// Device/Application/POUs/FB_MasterOperatorControl
FUNCTION_BLOCK FB_MasterOperatorControl
VAR_INPUT
    xAutoModeSelected     : BOOL;
    xEmergencyStopHealthy : BOOL;
    xFactoryIORunning     : BOOL;
    xManualModeSelected   : BOOL;
    xPlantFaulted         : BOOL;
    xResetPB              : BOOL;
    xStartPB              : BOOL;
    xStopCircuitHealthy   : BOOL;
END_VAR
VAR_OUTPUT
    xAutoModeActive   : BOOL;
    xAutoRun          : BOOL;
    xEnable           : BOOL;
    xManualModeActive : BOOL;
    xResetPulse       : BOOL;
    xResetRequired    : BOOL := TRUE;
    xRunLatched       : BOOL;
    xStopPending      : BOOL;
END_VAR
VAR
    fbResetEdge    : R_TRIG;
    fbStartEdge    : R_TRIG;
    xModeValid     : BOOL;
    xSafetyHealthy : BOOL;
END_VAR

// Convert the MASTER push buttons into one-scan events.
fbResetEdge(CLK := xResetPB);
fbStartEdge(CLK := xStartPB);

// Exactly one MASTER operating mode must be selected.
xModeValid :=
    xAutoModeSelected XOR xManualModeSelected;

xAutoModeActive :=
    xAutoModeSelected
    AND NOT xManualModeSelected;

xManualModeActive :=
    xManualModeSelected
    AND NOT xAutoModeSelected;

// MASTER safety availability.
// The ordinary Stop circuit is handled separately so Auto mode
// can finish its current transaction under controlled-stop logic.
xSafetyHealthy :=
    xEmergencyStopHealthy
    AND xFactoryIORunning
    AND xModeValid;

// One-scan default.
xResetPulse := FALSE;

// Immediate safety loss cancels all MASTER authority.
IF NOT xSafetyHealthy THEN
    xResetRequired := TRUE;
    xRunLatched := FALSE;
    xStopPending := FALSE;

// Reset has priority over a latched plant fault so that the
// coordinator can actually receive the reset pulse.
ELSIF fbResetEdge.Q AND xStopCircuitHealthy THEN
    xResetPulse := TRUE;
    xResetRequired := FALSE;
    xRunLatched := FALSE;
    xStopPending := FALSE;

// A plant fault removes the run latch and requires acknowledgement.
ELSIF xPlantFaulted THEN
    xResetRequired := TRUE;
    xRunLatched := FALSE;
    xStopPending := FALSE;

// MASTER Stop requests controlled completion in Auto mode.
ELSIF NOT xStopCircuitHealthy THEN
    IF xRunLatched THEN
        xStopPending := TRUE;
    END_IF

    xRunLatched := FALSE;

// Selecting Manual removes automatic authority.
// Local unit panels will receive authority in a later step.
ELSIF xManualModeActive THEN
    IF xRunLatched THEN
        xStopPending := TRUE;
    END_IF

    xRunLatched := FALSE;

// MASTER Start is accepted only in Auto after a valid reset.
ELSIF fbStartEdge.Q
    AND xAutoModeActive
    AND NOT xResetRequired
THEN
    xRunLatched := TRUE;
    xStopPending := FALSE;
END_IF

xAutoRun :=
    xAutoModeActive
    AND xRunLatched;

// Manual mode requires a healthy MASTER Stop circuit.
// Auto mode retains enable during a controlled-stop request.
xEnable :=
    xSafetyHealthy
    AND NOT xPlantFaulted
    AND NOT xResetRequired
    AND (
        xAutoModeActive
        OR xStopCircuitHealthy
    );

END_FUNCTION_BLOCK

// Device/Application/POUs/FB_PackoutCarrierStation
FUNCTION_BLOCK FB_PackoutCarrierStation
VAR_INPUT
    tStepTimeout      : TIME := T#30S;
    xCarrierReq       : BOOL;
    xDownstreamAck    : BOOL;
    xDownstreamReady  : BOOL;
    xEnable           : BOOL;
    xLoadComplete     : BOOL;
    xPalletAtLoad     : BOOL;
    xProductLoaded    : BOOL;
    xReset            : BOOL;
	xRun 			  : BOOL;
END_VAR
VAR_OUTPUT
    eState                    : E_PackoutCarrierState :=
                                    E_PackoutCarrierState.Stopped;
    uiFaultCode               : UINT;
    xBusy                     : BOOL;
    xCarrierConveyorCmd       : BOOL;
    xCarrierEmitterCmd        : BOOL;
    xCarrierInfeedConveyorCmd : BOOL;
    xCarrierReady             : BOOL;
    xFaulted                  : BOOL;
    xLoadAccepted             : BOOL;
    xLoadedCarrierReq         : BOOL;
    xReady                    : BOOL;
END_VAR
VAR
    ePreviousState 	   : E_PackoutCarrierState :=
                         E_PackoutCarrierState.Stopped;
	fbCarrierEmitPulse : TP;
    fbStepTimeout 	   : TON;
	xCarrierEmitIssued : BOOL;
    xStateChanged  	   : BOOL;
    xTimedState    	   : BOOL;
END_VAR

// Detect state transitions.
xStateChanged := eState <> ePreviousState;

fbCarrierEmitPulse(
    IN :=
        xEnable
        AND xRun
        AND NOT xCarrierEmitIssued
        AND
        (eState = E_PackoutCarrierState.FeedingCarrier)
        AND NOT xPalletAtLoad,
    PT := T#500MS
);

// Remember that this carrier has already been emitted.
// Preserve this latch across a controlled Stop.
IF fbCarrierEmitPulse.Q THEN
    xCarrierEmitIssued := TRUE;
END_IF

// Arrival proves that another carrier may be emitted later.
IF xPalletAtLoad THEN
    xCarrierEmitIssued := FALSE;
END_IF

xTimedState :=
    (eState = E_PackoutCarrierState.FeedingCarrier)
    OR
    (eState = E_PackoutCarrierState.TransferringCarrier)
    OR
    (eState =
        E_PackoutCarrierState.WaitingForDownstreamAckClear);

fbStepTimeout(
    IN :=
        xEnable
        AND xRun
        AND xTimedState
        AND NOT xStateChanged,
    PT := tStepTimeout
);

ePreviousState := eState;

// Safe physical-output defaults.
xCarrierConveyorCmd := FALSE;
xCarrierEmitterCmd := FALSE;
xCarrierInfeedConveyorCmd := FALSE;

IF xReset THEN
    eState := E_PackoutCarrierState.Stopped;
    ePreviousState := E_PackoutCarrierState.Stopped;
    uiFaultCode := 0;

ELSIF xEnable AND xRun THEN
    CASE eState OF

        E_PackoutCarrierState.Stopped:
            uiFaultCode := 0;
            eState :=
                E_PackoutCarrierState.WaitingForCarrierRequest;


        E_PackoutCarrierState.WaitingForCarrierRequest:
            IF xPalletAtLoad THEN
                eState :=
                    E_PackoutCarrierState.HoldingCarrierAtLoad;

            ELSIF xCarrierReq THEN
                eState :=
                    E_PackoutCarrierState.FeedingCarrier;
            END_IF


        E_PackoutCarrierState.FeedingCarrier:
            xCarrierConveyorCmd := TRUE;
            xCarrierEmitterCmd := fbCarrierEmitPulse.Q;
            xCarrierInfeedConveyorCmd := TRUE;

            IF xPalletAtLoad THEN
                eState :=
                    E_PackoutCarrierState.HoldingCarrierAtLoad;

            ELSIF fbStepTimeout.Q THEN
                uiFaultCode := 601;
                eState := E_PackoutCarrierState.Faulted;
            END_IF


        E_PackoutCarrierState.HoldingCarrierAtLoad:
            IF NOT xPalletAtLoad THEN
                IF xCarrierReq THEN
                    eState :=
                        E_PackoutCarrierState.FeedingCarrier;
                ELSE
                    eState :=
                        E_PackoutCarrierState
                            .WaitingForCarrierRequest;
                END_IF

            ELSIF xLoadComplete AND xProductLoaded THEN
                eState :=
                    E_PackoutCarrierState
                        .RequestingPlantStorage;
            END_IF


        E_PackoutCarrierState.RequestingPlantStorage:
            // Do not move until the loader has cleared its
            // LoadComplete request and Plant Storage is ready.
            IF NOT xLoadComplete AND xDownstreamReady THEN
                eState :=
                    E_PackoutCarrierState.TransferringCarrier;
            END_IF


        E_PackoutCarrierState.TransferringCarrier:
            xCarrierConveyorCmd := TRUE;

            IF xDownstreamAck THEN
                eState :=
                    E_PackoutCarrierState
                        .WaitingForDownstreamAckClear;

            ELSIF fbStepTimeout.Q THEN
                uiFaultCode := 602;
                eState := E_PackoutCarrierState.Faulted;
            END_IF


        E_PackoutCarrierState.WaitingForDownstreamAckClear:
            IF NOT xDownstreamAck THEN
                eState :=
                    E_PackoutCarrierState
                        .WaitingForCarrierRequest;

            ELSIF fbStepTimeout.Q THEN
                uiFaultCode := 603;
                eState := E_PackoutCarrierState.Faulted;
            END_IF


        E_PackoutCarrierState.Faulted:
            // Physical outputs remain at their safe defaults.


    ELSE
        uiFaultCode := 698;
        eState := E_PackoutCarrierState.Faulted;

    END_CASE
END_IF

// State-derived status and nonphysical handshakes.
xBusy :=
    (eState = E_PackoutCarrierState.FeedingCarrier)
    OR
    (eState = E_PackoutCarrierState.RequestingPlantStorage)
    OR
    (eState = E_PackoutCarrierState.TransferringCarrier)
    OR
    (eState =
        E_PackoutCarrierState.WaitingForDownstreamAckClear);

xCarrierReady :=
    xPalletAtLoad
    AND
    (eState = E_PackoutCarrierState.HoldingCarrierAtLoad);

xFaulted :=
    eState = E_PackoutCarrierState.Faulted;

xLoadAccepted :=
    xLoadComplete
    AND
    (eState =
        E_PackoutCarrierState.RequestingPlantStorage);

xLoadedCarrierReq :=
    NOT xLoadComplete
    AND
    (
        (eState =
            E_PackoutCarrierState.RequestingPlantStorage)
        OR
        (eState =
            E_PackoutCarrierState.TransferringCarrier)
    );

xReady :=
    xEnable
    AND xRun
	AND
    (
        (eState =
            E_PackoutCarrierState.WaitingForCarrierRequest)
        OR
        (eState =
            E_PackoutCarrierState.HoldingCarrierAtLoad)
    );

// Faults always remove physical commands.
IF xFaulted THEN
    xCarrierConveyorCmd := FALSE;
    xCarrierEmitterCmd := FALSE;
    xCarrierInfeedConveyorCmd := FALSE;
    xCarrierReady := FALSE;
    xReady := FALSE;
END_IF

END_FUNCTION_BLOCK

// Device/Application/POUs/FB_PackoutLoader
FUNCTION_BLOCK FB_PackoutLoader
VAR_INPUT
    tStepTimeout            : TIME := T#20S;
    xCarrierReady           : BOOL;
    xEnable                 : BOOL;
    xItemDetected           : BOOL;
    xLoadAccepted           : BOOL;
    xMovingX                : BOOL;
    xMovingZ                : BOOL;
    xProductAtPick          : BOOL;
    xProductLoaded          : BOOL;
    xProductTransferPermit  : BOOL;
    xReset                  : BOOL;
	xRun                    : BOOL;
END_VAR
VAR_OUTPUT
    diProductCount          : DINT;
    eState                  : E_PackoutLoaderState :=
                                  E_PackoutLoaderState.Stopped;
    uiFaultCode             : UINT;
    xBufferConveyor1Cmd     : BOOL;
    xBufferConveyor2Cmd     : BOOL;
    xBufferConveyor3Cmd     : BOOL;
    xBusy                   : BOOL;
    xCarrierReq             : BOOL;
    xFaulted                : BOOL;
    xGrabCmd                : BOOL;
    xLoadComplete           : BOOL;
    xMoveXCmd               : BOOL;
    xMoveZCmd               : BOOL;
    xPickConveyorCmd        : BOOL;
    xProductTransferAck     : BOOL;
    xProductTransferReady   : BOOL;
    xReady                  : BOOL;
END_VAR
VAR
    ePreviousState  : E_PackoutLoaderState :=
                          E_PackoutLoaderState.Stopped;
    fbGrabSettle     : TON;
	fbHomeStable     : TON;
    fbReleaseSettle  : TON;
    fbStepTimeout    : TON;
	xProductAccepted : BOOL;
    xSawXMotion      : BOOL;
    xSawZMotion      : BOOL;
    xStateChanged    : BOOL;
    xTimedState      : BOOL;
END_VAR

// Detect state transitions.
xStateChanged := eState <> ePreviousState;

IF xStateChanged THEN
    xSawXMotion := FALSE;
    xSawZMotion := FALSE;
END_IF

IF xMovingX THEN
    xSawXMotion := TRUE;
END_IF

IF xMovingZ THEN
    xSawZMotion := TRUE;
END_IF

fbHomeStable(
    IN :=
        xEnable
        AND xRun
        AND (eState = E_PackoutLoaderState.Homing)
        AND NOT xMovingX
        AND NOT xMovingZ,
    PT := T#500MS
);

xTimedState :=
    (eState <> E_PackoutLoaderState.Stopped)
    AND (eState <> E_PackoutLoaderState.WaitingForCarrier)
    AND (eState <> E_PackoutLoaderState.WaitingForProduct)
    AND
    (eState <>
        E_PackoutLoaderState.WaitingForLoadAcceptance)
    AND (eState <> E_PackoutLoaderState.Complete)
    AND (eState <> E_PackoutLoaderState.Faulted);

fbStepTimeout(
    IN :=
        xEnable
        AND xRun
        AND xTimedState
        AND NOT xStateChanged,
    PT := tStepTimeout
);

fbGrabSettle(
    IN :=
        xEnable
        AND xRun
        AND
        (eState = E_PackoutLoaderState.GrippingProduct),
    PT := T#500MS
);

fbReleaseSettle(
    IN :=
        xEnable
        AND xRun
        AND
        (eState = E_PackoutLoaderState.ReleasingProduct),
    PT := T#500MS
);

ePreviousState := eState;

// Safe defaults.
xBufferConveyor1Cmd := FALSE;
xBufferConveyor2Cmd := FALSE;
xBufferConveyor3Cmd := FALSE;
xBusy := FALSE;
xCarrierReq := FALSE;
xGrabCmd := FALSE;
xLoadComplete := FALSE;
xMoveXCmd := FALSE;
xMoveZCmd := FALSE;
xPickConveyorCmd := FALSE;
xProductTransferAck := FALSE;
xProductTransferReady := FALSE;
xReady := FALSE;

IF xReset THEN
    diProductCount := 0;
    eState := E_PackoutLoaderState.Stopped;
    ePreviousState := E_PackoutLoaderState.Stopped;
    uiFaultCode := 0;
    xFaulted := FALSE;
    xProductAccepted := FALSE;
    xSawXMotion := FALSE;
    xSawZMotion := FALSE;

ELSIF NOT xEnable THEN
    eState := E_PackoutLoaderState.Stopped;
    ePreviousState := E_PackoutLoaderState.Stopped;
    uiFaultCode := 0;
    xFaulted := FALSE;
    xProductAccepted := FALSE;
    xSawXMotion := FALSE;
    xSawZMotion := FALSE;

ELSIF xRun THEN
    CASE eState OF

        E_PackoutLoaderState.Stopped:
            xFaulted := FALSE;
            eState := E_PackoutLoaderState.Homing;


        E_PackoutLoaderState.Homing:
            // Both monostable axes return home with commands removed.
            IF fbHomeStable.Q THEN
                eState :=
                    E_PackoutLoaderState.WaitingForCarrier;

            ELSIF fbStepTimeout.Q THEN
                uiFaultCode := 501;
                xFaulted := TRUE;
                eState := E_PackoutLoaderState.Faulted;
            END_IF


        E_PackoutLoaderState.WaitingForCarrier:
            xCarrierReq := TRUE;
            xReady := TRUE;

            IF xCarrierReady THEN
                eState :=
                    E_PackoutLoaderState.WaitingForProduct;
            END_IF


        E_PackoutLoaderState.WaitingForProduct:
            xReady := TRUE;

            IF NOT xCarrierReady THEN
                eState :=
                    E_PackoutLoaderState.WaitingForCarrier;

            ELSE
                // A product already staged at the pick sensor
                // must not withdraw the loader's readiness.
                xProductTransferReady := NOT xProductLoaded;

                IF xProductTransferPermit THEN
                    xBufferConveyor1Cmd := NOT xProductAtPick;
                    xBufferConveyor2Cmd := NOT xProductAtPick;
                    xBufferConveyor3Cmd := NOT xProductAtPick;
                    xPickConveyorCmd := NOT xProductAtPick;

                    IF xProductAtPick THEN
                        xProductAccepted := TRUE;
                        eState :=
                            E_PackoutLoaderState.MovingToProduct;
                    END_IF
                END_IF
            END_IF


        E_PackoutLoaderState.MovingToProduct:
            xBusy := TRUE;
            xMoveXCmd := TRUE;

            IF xSawXMotion AND NOT xMovingX THEN
                eState :=
                    E_PackoutLoaderState.LoweringToProduct;

            ELSIF fbStepTimeout.Q THEN
                uiFaultCode := 503;
                xFaulted := TRUE;
                eState := E_PackoutLoaderState.Faulted;
            END_IF


        E_PackoutLoaderState.LoweringToProduct:
            xBusy := TRUE;
            xMoveXCmd := TRUE;
            xMoveZCmd := TRUE;

            IF xSawZMotion AND NOT xMovingZ THEN
                eState :=
                    E_PackoutLoaderState.GrippingProduct;

            ELSIF fbStepTimeout.Q THEN
                uiFaultCode := 504;
                xFaulted := TRUE;
                eState := E_PackoutLoaderState.Faulted;
            END_IF


        E_PackoutLoaderState.GrippingProduct:
            xBusy := TRUE;
            xGrabCmd := TRUE;
            xMoveXCmd := TRUE;
            xMoveZCmd := TRUE;

            IF fbGrabSettle.Q AND xItemDetected THEN
                eState :=
                    E_PackoutLoaderState.RaisingProduct;

            ELSIF fbStepTimeout.Q THEN
                uiFaultCode := 505;
                xFaulted := TRUE;
                eState := E_PackoutLoaderState.Faulted;
            END_IF


        E_PackoutLoaderState.RaisingProduct:
            xBusy := TRUE;
            xGrabCmd := TRUE;
            xMoveXCmd := TRUE;

            IF xSawZMotion AND NOT xMovingZ THEN
                eState :=
                    E_PackoutLoaderState.MovingToCarrier;

            ELSIF fbStepTimeout.Q THEN
                uiFaultCode := 506;
                xFaulted := TRUE;
                eState := E_PackoutLoaderState.Faulted;
            END_IF


        E_PackoutLoaderState.MovingToCarrier:
            xBusy := TRUE;
            xGrabCmd := TRUE;

            // Removing the X command retracts the monostable
            // horizontal axis towards the carrier.
            IF xSawXMotion AND NOT xMovingX THEN
                eState :=
                    E_PackoutLoaderState.LoweringToCarrier;

            ELSIF fbStepTimeout.Q THEN
                uiFaultCode := 507;
                xFaulted := TRUE;
                eState := E_PackoutLoaderState.Faulted;
            END_IF


        E_PackoutLoaderState.LoweringToCarrier:
            xBusy := TRUE;
            xGrabCmd := TRUE;
            xMoveZCmd := TRUE;

            IF xSawZMotion AND NOT xMovingZ THEN
                eState :=
                    E_PackoutLoaderState.ReleasingProduct;

            ELSIF fbStepTimeout.Q THEN
                uiFaultCode := 508;
                xFaulted := TRUE;
                eState := E_PackoutLoaderState.Faulted;
            END_IF


        E_PackoutLoaderState.ReleasingProduct:
            xBusy := TRUE;
            xMoveZCmd := TRUE;

            IF fbReleaseSettle.Q AND NOT xItemDetected THEN
                eState :=
                    E_PackoutLoaderState.RaisingFromCarrier;

            ELSIF fbStepTimeout.Q THEN
                uiFaultCode := 509;
                xFaulted := TRUE;
                eState := E_PackoutLoaderState.Faulted;
            END_IF


        E_PackoutLoaderState.RaisingFromCarrier:
            xBusy := TRUE;

            IF xSawZMotion AND NOT xMovingZ THEN
                eState :=
                    E_PackoutLoaderState.ReturningHome;

            ELSIF fbStepTimeout.Q THEN
                uiFaultCode := 510;
                xFaulted := TRUE;
                eState := E_PackoutLoaderState.Faulted;
            END_IF


        E_PackoutLoaderState.ReturningHome:
            xBusy := TRUE;

            IF NOT xMovingX AND NOT xMovingZ THEN
                eState :=
                    E_PackoutLoaderState.VerifyingLoad;

            ELSIF fbStepTimeout.Q THEN
                uiFaultCode := 511;
                xFaulted := TRUE;
                eState := E_PackoutLoaderState.Faulted;
            END_IF


        E_PackoutLoaderState.VerifyingLoad:
            xBusy := TRUE;

            IF xCarrierReady AND xProductLoaded THEN
                diProductCount := diProductCount + 1;
                eState :=
                    E_PackoutLoaderState
                        .WaitingForLoadAcceptance;

            ELSIF fbStepTimeout.Q THEN
                uiFaultCode := 512;
                xFaulted := TRUE;
                eState := E_PackoutLoaderState.Faulted;
            END_IF


        E_PackoutLoaderState.WaitingForLoadAcceptance:
            xBusy := TRUE;
            xLoadComplete := TRUE;

            IF xLoadAccepted THEN
                eState := E_PackoutLoaderState.Complete;
            END_IF


        E_PackoutLoaderState.Complete:
            // Wait for the carrier station to clear acknowledgement.
            IF NOT xLoadAccepted THEN
                eState :=
                    E_PackoutLoaderState.WaitingForCarrier;
            END_IF


        E_PackoutLoaderState.Faulted:
            xFaulted := TRUE;


    ELSE
        uiFaultCode := 599;
        xFaulted := TRUE;
        eState := E_PackoutLoaderState.Faulted;

    END_CASE
END_IF

// A controlled Stop preserves the current transaction.
// The monostable axes retain the command appropriate to the
// current sequence state.
IF xEnable AND NOT xRun AND NOT xFaulted THEN
    xBusy :=
        (eState = E_PackoutLoaderState.MovingToProduct)
        OR (eState = E_PackoutLoaderState.LoweringToProduct)
        OR (eState = E_PackoutLoaderState.GrippingProduct)
        OR (eState = E_PackoutLoaderState.RaisingProduct)
        OR (eState = E_PackoutLoaderState.MovingToCarrier)
        OR (eState = E_PackoutLoaderState.LoweringToCarrier)
        OR (eState = E_PackoutLoaderState.ReleasingProduct)
        OR (eState = E_PackoutLoaderState.RaisingFromCarrier)
        OR (eState = E_PackoutLoaderState.ReturningHome)
        OR (eState = E_PackoutLoaderState.VerifyingLoad)
        OR
        (eState =
            E_PackoutLoaderState.WaitingForLoadAcceptance);

    xGrabCmd :=
        (eState = E_PackoutLoaderState.GrippingProduct)
        OR (eState = E_PackoutLoaderState.RaisingProduct)
        OR (eState = E_PackoutLoaderState.MovingToCarrier)
        OR (eState = E_PackoutLoaderState.LoweringToCarrier);

    xLoadComplete :=
        eState =
            E_PackoutLoaderState.WaitingForLoadAcceptance;

    xMoveXCmd :=
        (eState = E_PackoutLoaderState.MovingToProduct)
        OR (eState = E_PackoutLoaderState.LoweringToProduct)
        OR (eState = E_PackoutLoaderState.GrippingProduct)
        OR (eState = E_PackoutLoaderState.RaisingProduct);

    xMoveZCmd :=
        (eState = E_PackoutLoaderState.LoweringToProduct)
        OR (eState = E_PackoutLoaderState.GrippingProduct)
        OR (eState = E_PackoutLoaderState.LoweringToCarrier)
        OR (eState = E_PackoutLoaderState.ReleasingProduct);
END_IF

// Hold acknowledgement until the coordinator removes its permit.
xProductTransferAck := xProductAccepted;

IF xProductAccepted
    AND xRun
    AND NOT xProductTransferPermit
THEN
    xProductAccepted := FALSE;
    xProductTransferAck := FALSE;
END_IF

// Faults remove every command and handshake.
IF xFaulted THEN
    xBufferConveyor1Cmd := FALSE;
    xBufferConveyor2Cmd := FALSE;
    xBufferConveyor3Cmd := FALSE;
    xCarrierReq := FALSE;
    xGrabCmd := FALSE;
    xLoadComplete := FALSE;
    xMoveXCmd := FALSE;
    xMoveZCmd := FALSE;
    xPickConveyorCmd := FALSE;
    xProductAccepted := FALSE;
    xProductTransferAck := FALSE;
    xProductTransferReady := FALSE;
    xReady := FALSE;
END_IF

END_FUNCTION_BLOCK

// Device/Application/POUs/FB_PairDiverter
FUNCTION_BLOCK FB_PairDiverter
VAR_INPUT
	tLidPositionTime 		   : TIME := T#300MS;
    tStepTimeout               : TIME := T#15S;
    xAssemblyBaseAtPlace       : BOOL;
    xAssemblyLidAtPlace        : BOOL;
    xCountDetected             : BOOL;
    xEnable                    : BOOL;
    xPartAtPusher              : BOOL;
    xPusherAtBack              : BOOL;
    xPusherAtFront             : BOOL;
    xReset                     : BOOL;
	xRun					   : BOOL;
    xTransferPermit            : BOOL;
END_VAR
VAR_OUTPUT
    diDetectionCount       : DINT;
    eState                 : E_PairDiverterState := E_PairDiverterState.Idle;
    uiFaultCode            : UINT;
    xBaseCurveConveyorCmd  : BOOL;
    xBasesOutfeedCmd       : BOOL;
    xComplete              : BOOL;
    xFaulted               : BOOL;
    xInfeedConveyorCmd     : BOOL;
    xLidsOutfeedCmd        : BOOL;
    xPusherCmd             : BOOL;
    xPusherZoneConveyorCmd : BOOL;
END_VAR
VAR
    ePreviousState     : E_PairDiverterState := E_PairDiverterState.Idle;
    fbCountEdge        : R_TRIG;
	fbLidPositionDelay : TON;
    fbLidReleaseDelay  : TON;
    fbStepTimeout      : TON;
    xStateChanged      : BOOL;
    xTimeoutActive     : BOOL;
END_VAR

// Count products crossing the dedicated total-count sensor.
fbCountEdge(CLK := xCountDetected);

// Release the lid two seconds after releasing the base.
fbLidReleaseDelay(
    IN :=
        xRun
        AND (eState = E_PairDiverterState.ReleasingBase),
    PT := T#2S
);

// Move the detected lid from the approach sensor to the
// centreline of the pusher before extending the pusher.
fbLidPositionDelay(
    IN :=
        xRun
        AND
        (eState = E_PairDiverterState.PositioningLid),
    PT := tLidPositionTime
);

// Reset the step timeout whenever the state changes.
xStateChanged := eState <> ePreviousState;

xTimeoutActive :=
    (eState <> E_PairDiverterState.Idle)
    AND (eState <> E_PairDiverterState.Complete)
    AND (eState <> E_PairDiverterState.Faulted)
    AND NOT xStateChanged;

fbStepTimeout(
    IN := xRun AND xTimeoutActive,
    PT := tStepTimeout
);

ePreviousState := eState;

// Default every command and pulse off.
xBaseCurveConveyorCmd := FALSE;
xBasesOutfeedCmd := FALSE;
xComplete := FALSE;
xInfeedConveyorCmd := FALSE;
xLidsOutfeedCmd := FALSE;
xPusherCmd := FALSE;
xPusherZoneConveyorCmd := FALSE;

IF xReset THEN
    diDetectionCount := 0;
    eState := E_PairDiverterState.Idle;
    ePreviousState := E_PairDiverterState.Idle;
    uiFaultCode := 0;
    xFaulted := FALSE;

ELSIF NOT xEnable THEN
    eState := E_PairDiverterState.Idle;
    ePreviousState := E_PairDiverterState.Idle;
    uiFaultCode := 0;
    xFaulted := FALSE;

ELSIF xRun THEN
    IF fbCountEdge.Q THEN
        diDetectionCount := diDetectionCount + 1;
    END_IF

    CASE eState OF

        E_PairDiverterState.Idle:
            xFaulted := FALSE;

            IF xTransferPermit
                AND NOT xAssemblyBaseAtPlace
                AND NOT xAssemblyLidAtPlace
                AND NOT xPartAtPusher
                AND xPusherAtBack
            THEN
                eState := E_PairDiverterState.ReleasingBase;
            END_IF


        E_PairDiverterState.ReleasingBase:
            // Start the base route first.
            xBaseCurveConveyorCmd := TRUE;
            xBasesOutfeedCmd := TRUE;
            xInfeedConveyorCmd := TRUE;
            xPusherZoneConveyorCmd := TRUE;

            IF fbLidReleaseDelay.Q THEN
                eState := E_PairDiverterState.ReleasingLid;

            ELSIF fbStepTimeout.Q THEN
                uiFaultCode := 301;
                xFaulted := TRUE;
                eState := E_PairDiverterState.Faulted;
            END_IF


        E_PairDiverterState.ReleasingLid:
            // Keep the base moving and start the lid two seconds behind.
            xBaseCurveConveyorCmd := NOT xAssemblyBaseAtPlace;
            xBasesOutfeedCmd := NOT xAssemblyBaseAtPlace;
            xInfeedConveyorCmd := TRUE;
            xLidsOutfeedCmd := TRUE;
            xPusherZoneConveyorCmd := TRUE;

            // The first item reaching the pusher is the base.
            // It must pass without a pusher command.
            IF xPartAtPusher THEN
                eState := E_PairDiverterState.PassingBase;

            ELSIF fbStepTimeout.Q THEN
                uiFaultCode := 302;
                xFaulted := TRUE;
                eState := E_PairDiverterState.Faulted;
            END_IF


        E_PairDiverterState.PassingBase:
            xBaseCurveConveyorCmd := NOT xAssemblyBaseAtPlace;
            xBasesOutfeedCmd := NOT xAssemblyBaseAtPlace;
            xInfeedConveyorCmd := TRUE;
            xLidsOutfeedCmd := TRUE;
            xPusherZoneConveyorCmd := TRUE;

            // The base has passed once it clears the pusher sensor.
            IF NOT xPartAtPusher THEN
                eState := E_PairDiverterState.WaitingForLidAtPusher;

            ELSIF fbStepTimeout.Q THEN
                uiFaultCode := 303;
                xFaulted := TRUE;
                eState := E_PairDiverterState.Faulted;
            END_IF


        E_PairDiverterState.WaitingForLidAtPusher:
            xBaseCurveConveyorCmd := NOT xAssemblyBaseAtPlace;
            xBasesOutfeedCmd := NOT xAssemblyBaseAtPlace;
            xInfeedConveyorCmd := TRUE;
            xLidsOutfeedCmd := TRUE;
            xPusherZoneConveyorCmd := TRUE;

            IF xPartAtPusher THEN
                // The lid must be the second/even detected product.
                IF (diDetectionCount > 0)
                    AND ((diDetectionCount MOD 2) = 0)
                THEN
                    eState := E_PairDiverterState.PositioningLid;
                ELSE
                    uiFaultCode := 312;
                    xFaulted := TRUE;
                    eState := E_PairDiverterState.Faulted;
                END_IF

            ELSIF fbStepTimeout.Q THEN
                uiFaultCode := 304;
                xFaulted := TRUE;
                eState := E_PairDiverterState.Faulted;
            END_IF


        E_PairDiverterState.PositioningLid:
		// The approach sensor has already latched the lid's arrival.
		// Index it forwards briefly until centred on the pusher.
		xBaseCurveConveyorCmd := NOT xAssemblyBaseAtPlace;
		xBasesOutfeedCmd := NOT xAssemblyBaseAtPlace;
		xInfeedConveyorCmd := NOT fbLidPositionDelay.Q;
		xPusherZoneConveyorCmd := NOT fbLidPositionDelay.Q;
	
		IF fbLidPositionDelay.Q AND xPusherAtBack THEN
			eState := E_PairDiverterState.PushingLid;
	
		ELSIF fbStepTimeout.Q THEN
			uiFaultCode := 305;
			xFaulted := TRUE;
			eState := E_PairDiverterState.Faulted;
    	END_IF


        E_PairDiverterState.PushingLid:
            xBaseCurveConveyorCmd := NOT xAssemblyBaseAtPlace;
            xBasesOutfeedCmd := NOT xAssemblyBaseAtPlace;
            xPusherCmd := TRUE;

            IF xPusherAtFront THEN
                eState := E_PairDiverterState.WaitingForPartsAtPlace;

            ELSIF fbStepTimeout.Q THEN
                uiFaultCode := 306;
                xFaulted := TRUE;
                eState := E_PairDiverterState.Faulted;
            END_IF


        E_PairDiverterState.WaitingForPartsAtPlace:
            // Removing the command retracts the monostable pusher.
            xBaseCurveConveyorCmd := NOT xAssemblyBaseAtPlace;
            xBasesOutfeedCmd := NOT xAssemblyBaseAtPlace;
            xPusherZoneConveyorCmd := NOT xAssemblyLidAtPlace;

            IF xAssemblyBaseAtPlace
                AND xAssemblyLidAtPlace
                AND xPusherAtBack
            THEN
                eState := E_PairDiverterState.Complete;

            ELSIF fbStepTimeout.Q THEN
                uiFaultCode := 307;
                xFaulted := TRUE;
                eState := E_PairDiverterState.Faulted;
            END_IF


        E_PairDiverterState.Complete:
            xComplete := TRUE;

            IF NOT xTransferPermit THEN
                eState := E_PairDiverterState.Idle;
            END_IF


        E_PairDiverterState.Faulted:
            xFaulted := TRUE;


    ELSE
        uiFaultCode := 399;
        xFaulted := TRUE;
        eState := E_PairDiverterState.Faulted;

    END_CASE
END_IF

// A fault removes all physical commands.
IF xFaulted THEN
    xBaseCurveConveyorCmd := FALSE;
    xBasesOutfeedCmd := FALSE;
    xInfeedConveyorCmd := FALSE;
    xLidsOutfeedCmd := FALSE;
    xPusherCmd := FALSE;
    xPusherZoneConveyorCmd := FALSE;
END_IF

END_FUNCTION_BLOCK

// Device/Application/POUs/FB_TransferCoordinator
FUNCTION_BLOCK FB_TransferCoordinator
VAR_INPUT
    tTransferTimeout : TIME := T#20S;
    xAck             : BOOL;
    xEnable          : BOOL;
    xReady           : BOOL;
    xReq             : BOOL;
    xReset           : BOOL;
	xRun 			 : BOOL;
END_VAR
VAR
    fbTransferTimeout : TON;
    xTimeoutEnable    : BOOL;
END_VAR
VAR_OUTPUT
    eState      : E_TransferState := E_TransferState.Idle;
    uiFaultCode : UINT;
    xComplete   : BOOL;
    xFaulted    : BOOL;
    xPermit     : BOOL;
END_VAR

// Default pulse outputs.
xComplete := FALSE;

// A controlled zone Stop removes permission while preserving state.
xPermit := FALSE;

// The timeout runs during every active handshake stage.
xTimeoutEnable :=
    (eState = E_TransferState.WaitingForReady)
    OR (eState = E_TransferState.Transferring)
    OR (eState = E_TransferState.WaitingForRequestClear);

fbTransferTimeout(
    IN := xRun AND xTimeoutEnable,
    PT := tTransferTimeout
);

// Reset has priority over every state.
IF xReset THEN
    eState := E_TransferState.Idle;
    uiFaultCode := 0;
    xFaulted := FALSE;
    xPermit := FALSE;

ELSIF NOT xEnable THEN
    eState := E_TransferState.Idle;
    uiFaultCode := 0;
    xFaulted := FALSE;
    xPermit := FALSE;

ELSIF xRun THEN
    CASE eState OF

        E_TransferState.Idle:
            xPermit := FALSE;

            IF xReq THEN
                eState := E_TransferState.WaitingForReady;
            END_IF


        E_TransferState.WaitingForReady:
            xPermit := FALSE;

            IF xReady THEN
                xPermit := TRUE;
                eState := E_TransferState.Transferring;

            ELSIF fbTransferTimeout.Q THEN
                uiFaultCode := 201;
                xFaulted := TRUE;
                eState := E_TransferState.Faulted;
            END_IF


        E_TransferState.Transferring:
            xPermit := TRUE;

            IF xAck THEN
                xPermit := FALSE;
                eState := E_TransferState.WaitingForRequestClear;

            ELSIF fbTransferTimeout.Q THEN
                uiFaultCode := 202;
                xFaulted := TRUE;
                xPermit := FALSE;
                eState := E_TransferState.Faulted;
            END_IF


        E_TransferState.WaitingForRequestClear:
            xPermit := FALSE;

            IF NOT xReq THEN
                xComplete := TRUE;
                eState := E_TransferState.Idle;

            ELSIF fbTransferTimeout.Q THEN
                uiFaultCode := 203;
                xFaulted := TRUE;
                eState := E_TransferState.Faulted;
            END_IF


        E_TransferState.Faulted:
            xPermit := FALSE;
            xFaulted := TRUE;


    ELSE
        uiFaultCode := 299;
        xFaulted := TRUE;
        xPermit := FALSE;
        eState := E_TransferState.Faulted;

    END_CASE
END_IF

END_FUNCTION_BLOCK

// Device/Application/POUs/FB_PlantCoordinator
FUNCTION_BLOCK FB_PlantCoordinator
VAR_INPUT
    xAnyFault                : BOOL;
    xAutoRun                 : BOOL;
    xBatchStorageReady       : BOOL;
    xEnable                  : BOOL;
    xPairTransferComplete    : BOOL;
    xProductTransferComplete : BOOL;
    xRackCommitAck           : BOOL;
    xRackReservationValid    : BOOL;
    xReset                   : BOOL;
END_VAR
VAR_OUTPUT
    eProductionPhase       : E_ProductionPhase := E_ProductionPhase.Idle;
    eState                 : E_PlantState := E_PlantState.Stopped;
    uiFaultCode            : UINT;
    xAllowNewPair          : BOOL;
    xFaulted               : BOOL;
    xPairTransferEnable    : BOOL;
    xProductTransferEnable : BOOL;
    xRecoveryRequired      : BOOL;
    xRunning               : BOOL;
    xStopPending           : BOOL;
END_VAR

// Safe defaults recalculated on every scan.
xAllowNewPair := FALSE;
xFaulted := FALSE;
xPairTransferEnable := FALSE;
xProductTransferEnable := FALSE;
xRecoveryRequired := FALSE;
xRunning := FALSE;

// Reset always returns the plant coordinator to a known state.
IF xReset THEN
    eProductionPhase := E_ProductionPhase.Idle;
    eState := E_PlantState.Stopped;
    uiFaultCode := 0;
    xStopPending := FALSE;

ELSIF xAnyFault THEN
    uiFaultCode := 401;
    xFaulted := TRUE;
    xStopPending := FALSE;
    eState := E_PlantState.Faulted;

ELSE
    CASE eState OF

        E_PlantState.Stopped:
            eProductionPhase := E_ProductionPhase.Idle;
            uiFaultCode := 0;
            xStopPending := FALSE;

            IF xEnable AND xAutoRun THEN
                eState := E_PlantState.Starting;
            END_IF


        E_PlantState.Starting:
            xRunning := TRUE;
            eProductionPhase := E_ProductionPhase.ReservingStorage;

            // Do not begin production without both downstream
            // availability and a reserved rack destination.
            IF xRackReservationValid AND xBatchStorageReady THEN
                eProductionPhase := E_ProductionPhase.ProducingPair;
                eState := E_PlantState.Running;

            ELSIF NOT xEnable THEN
                eState := E_PlantState.Stopped;
            END_IF


        E_PlantState.Running:
            xRunning := TRUE;

            // Releasing Auto Run requests a controlled stop.
            // The current transaction is allowed to finish.
            IF NOT xAutoRun THEN
                xStopPending := TRUE;
            END_IF

            CASE eProductionPhase OF

                E_ProductionPhase.Idle:
                    // No active product exists, so a requested stop
                    // can complete immediately.
                    IF xStopPending THEN
                        eState := E_PlantState.Stopping;

                    ELSIF xRackReservationValid
                        AND xBatchStorageReady
                    THEN
                        eProductionPhase :=
                            E_ProductionPhase.ProducingPair;
                    END_IF


                E_ProductionPhase.ReservingStorage:
                    IF xRackReservationValid
                        AND xBatchStorageReady
                    THEN
                        eProductionPhase :=
                            E_ProductionPhase.ProducingPair;
                    END_IF


                E_ProductionPhase.ProducingPair:
                    xAllowNewPair := NOT xStopPending;
                    xPairTransferEnable := TRUE;

                    IF xPairTransferComplete THEN
                        eProductionPhase :=
                            E_ProductionPhase.Assembling;
                    END_IF


                E_ProductionPhase.Assembling:
                    xProductTransferEnable := TRUE;

                    IF xProductTransferComplete THEN
                        eProductionPhase :=
                            E_ProductionPhase.WaitingForPackout;
                    END_IF


                E_ProductionPhase.WaitingForPackout:
                    // Packout/P9 detail is added when those equipment
                    // FBs are integrated. For now, downstream becoming
                    // busy proves that the loaded carrier was accepted.
                    IF NOT xBatchStorageReady THEN
                        eProductionPhase :=
                            E_ProductionPhase.Batching;
                    END_IF


                E_ProductionPhase.Batching:
                    // The rack commit confirms that the tank/storage
                    // transaction ultimately completed.
                    IF xRackCommitAck THEN
                        eProductionPhase :=
                            E_ProductionPhase.Complete;
                    END_IF


                E_ProductionPhase.Storing:
                    IF xRackCommitAck THEN
                        eProductionPhase :=
                            E_ProductionPhase.Complete;
                    END_IF


                E_ProductionPhase.Complete:
                    IF xStopPending THEN
                        eState := E_PlantState.Stopping;
                    ELSE
                        eProductionPhase :=
                            E_ProductionPhase.ReservingStorage;
                        eState := E_PlantState.Starting;
                    END_IF


            ELSE
                uiFaultCode := 402;
                eState := E_PlantState.Faulted;

            END_CASE


        E_PlantState.Stopping:
            // This state is reached only after the active load has
            // completed or when no load was active.
            eProductionPhase := E_ProductionPhase.Idle;
            xStopPending := FALSE;
            eState := E_PlantState.Stopped;


        E_PlantState.Faulted:
            xFaulted := TRUE;


        E_PlantState.RecoveryRequired:
            xRecoveryRequired := TRUE;


    ELSE
        uiFaultCode := 499;
        eState := E_PlantState.Faulted;

    END_CASE
END_IF

// Loss of the overall enable removes all permissions immediately.
IF NOT xEnable THEN
    xAllowNewPair := FALSE;
    xPairTransferEnable := FALSE;
    xProductTransferEnable := FALSE;
    xRunning := FALSE;

    IF eState <> E_PlantState.Faulted THEN
        eProductionPhase := E_ProductionPhase.Idle;
        eState := E_PlantState.Stopped;
        xStopPending := FALSE;
    END_IF
END_IF

END_FUNCTION_BLOCK

// Device/Application/POUs/FB_TwinCellUnit
FUNCTION_BLOCK FB_TwinCellUnit
VAR_INPUT
    xEnable                         : BOOL;
    xPairAccepted                   : BOOL;
	xProductionRequest 				: BOOL;
    xReset                          : BOOL;
    xRun                            : BOOL;
    xTwinCellBasesCenterBusy        : BOOL;
    xTwinCellBasesCenterHasError    : BOOL;
    xTwinCellBasesCenterOpened      : BOOL;
    xTwinCellBasesEntryDetected     : BOOL;
    xTwinCellBasesExitDetected      : BOOL;
    xTwinCellLidsCenterBusy         : BOOL;
    xTwinCellLidsCenterHasError     : BOOL;
    xTwinCellLidsCenterOpened       : BOOL;
    xTwinCellLidsEntryDetected      : BOOL;
    xTwinCellLidsExitDetected       : BOOL;
END_VAR
VAR_OUTPUT
    diBasesCount               : DINT;
    diLidsCount                : DINT;
    diPairCount                : DINT;
    uiBasesFaultCode           : UINT;
    uiFaultCode                : UINT;
    uiLidsFaultCode            : UINT;
    xBasesBusy                 : BOOL;
    xBasesCenterProduceCmd     : BOOL;
    xBasesCenterResetCmd       : BOOL;
    xBasesCenterStartCmd       : BOOL;
    xBasesCenterStopCmd        : BOOL;
    xBasesEmitterCmd           : BOOL;
    xBasesExitConveyor1Cmd     : BOOL;
    xBasesExitConveyor2Cmd     : BOOL;
    xBasesFaulted              : BOOL;
    xBasesRawConveyorCmd       : BOOL;
    xBasesReady                : BOOL;
    xBusy                      : BOOL;
    xFaulted                   : BOOL;
    xLidsBusy                  : BOOL;
    xLidsCenterProduceCmd      : BOOL;
    xLidsCenterResetCmd        : BOOL;
    xLidsCenterStartCmd        : BOOL;
    xLidsCenterStopCmd         : BOOL;
    xLidsEmitterCmd            : BOOL;
    xLidsExitConveyor1Cmd      : BOOL;
    xLidsExitConveyor2Cmd      : BOOL;
    xLidsFaulted               : BOOL;
    xLidsRawConveyorCmd        : BOOL;
    xLidsReady                 : BOOL;
    xPairReq                   : BOOL;
    xReady                     : BOOL;
END_VAR
VAR
    fbBasesMachiningCell : FB_MachiningCell;
    fbLidsMachiningCell  : FB_MachiningCell;
    xPairPending         : BOOL;
    xWaitForExitClear    : BOOL;
END_VAR

// Twin Cell owns both machining-cell instances.
fbBasesMachiningCell(
	tProcessTimeout := T#90S,
    xAtEntry := xTwinCellBasesEntryDetected,
    xAtExit := xTwinCellBasesExitDetected,
    xCenterBusy := xTwinCellBasesCenterBusy,
    xCenterHasError := xTwinCellBasesCenterHasError,
    xCenterOpened := xTwinCellBasesCenterOpened,
    xEnable := xEnable,
    xProduceLids := FALSE,
	xRequest := xProductionRequest,
    xReset := xReset,
    xRun := xRun
);

fbLidsMachiningCell(
	tProcessTimeout := T#90S,
    xAtEntry := xTwinCellLidsEntryDetected,
    xAtExit := xTwinCellLidsExitDetected,
    xCenterBusy := xTwinCellLidsCenterBusy,
    xCenterHasError := xTwinCellLidsCenterHasError,
    xCenterOpened := xTwinCellLidsCenterOpened,
    xEnable := xEnable,
    xProduceLids := TRUE,
	xRequest := xProductionRequest,
    xReset := xReset,
    xRun := xRun
);

// Publish both machining-cell boundaries.
diBasesCount := fbBasesMachiningCell.diCount;
diLidsCount := fbLidsMachiningCell.diCount;

uiBasesFaultCode := fbBasesMachiningCell.uiFaultCode;
uiLidsFaultCode := fbLidsMachiningCell.uiFaultCode;

xBasesBusy := fbBasesMachiningCell.xBusy;
xBasesCenterProduceCmd :=
    fbBasesMachiningCell.xCenterProduceCmd;
xBasesCenterResetCmd :=
    fbBasesMachiningCell.xCenterResetCmd;
xBasesCenterStartCmd :=
    fbBasesMachiningCell.xCenterStartCmd;
xBasesCenterStopCmd :=
    fbBasesMachiningCell.xCenterStopCmd;
xBasesEmitterCmd := fbBasesMachiningCell.xEmitterCmd;
xBasesExitConveyor1Cmd :=
    fbBasesMachiningCell.xExitConveyor1Cmd;
xBasesExitConveyor2Cmd :=
    fbBasesMachiningCell.xExitConveyor2Cmd;
xBasesFaulted := fbBasesMachiningCell.xFaulted;
xBasesRawConveyorCmd :=
    fbBasesMachiningCell.xRawConveyorCmd;
xBasesReady := fbBasesMachiningCell.xReady;

xLidsBusy := fbLidsMachiningCell.xBusy;
xLidsCenterProduceCmd :=
    fbLidsMachiningCell.xCenterProduceCmd;
xLidsCenterResetCmd :=
    fbLidsMachiningCell.xCenterResetCmd;
xLidsCenterStartCmd :=
    fbLidsMachiningCell.xCenterStartCmd;
xLidsCenterStopCmd :=
    fbLidsMachiningCell.xCenterStopCmd;
xLidsEmitterCmd := fbLidsMachiningCell.xEmitterCmd;
xLidsExitConveyor1Cmd :=
    fbLidsMachiningCell.xExitConveyor1Cmd;
xLidsExitConveyor2Cmd :=
    fbLidsMachiningCell.xExitConveyor2Cmd;
xLidsFaulted := fbLidsMachiningCell.xFaulted;
xLidsRawConveyorCmd :=
    fbLidsMachiningCell.xRawConveyorCmd;
xLidsReady := fbLidsMachiningCell.xReady;

// =============================================================
// UNIT STATUS DEFAULTS
// =============================================================

xFaulted := xBasesFaulted OR xLidsFaulted;

xBusy :=
    xBasesBusy
    OR xLidsBusy
    OR xPairPending
    OR xWaitForExitClear;

xPairReq := FALSE;
xReady := FALSE;

// Prefix the child fault code so its source remains identifiable.
IF xBasesFaulted THEN
    uiFaultCode := UINT#1000 + uiBasesFaultCode;

ELSIF xLidsFaulted THEN
    uiFaultCode := UINT#2000 + uiLidsFaultCode;

ELSE
    uiFaultCode := 0;
END_IF

// =============================================================
// RESET, FAULT AND RUN PRIORITIES
// =============================================================

// Reset clears both child faults, the pending transaction
// and the completed-pair count.
IF xReset THEN
    diPairCount := 0;
    uiFaultCode := 0;
    xFaulted := FALSE;
    xPairPending := FALSE;
    xWaitForExitClear := FALSE;

// A child-cell fault abandons any untransferred pair.
ELSIF xFaulted THEN
    xPairPending := FALSE;
    xWaitForExitClear := FALSE;

// Disabling the unit abandons any untransferred request,
// but retains the production counts.
ELSIF NOT xEnable THEN
    xPairPending := FALSE;
    xWaitForExitClear := FALSE;

// A controlled Stop freezes transaction memory.
ELSIF xRun THEN

    // After a pair is accepted, require both P10 exit sensors
    // to clear before recognising another completed pair.
    IF xWaitForExitClear THEN
		IF NOT fbBasesMachiningCell.xDone
			AND NOT fbLidsMachiningCell.xDone
		THEN
			xWaitForExitClear := FALSE;
		END_IF
	
	ELSIF NOT xPairPending
		AND fbBasesMachiningCell.xDone
		AND fbLidsMachiningCell.xDone
	THEN
		xPairPending := TRUE;
	END_IF

    // Acceptance means the P10-to-P11 transfer completed.
    IF xPairPending AND xPairAccepted THEN
        diPairCount := diPairCount + 1;
        xPairPending := FALSE;
        xWaitForExitClear := TRUE;
    END_IF

    xPairReq := xPairPending;

    xBusy :=
        xBasesBusy
        OR xLidsBusy
        OR xPairPending
        OR xWaitForExitClear;

    xReady :=
        xBasesReady
        AND xLidsReady
        AND NOT xPairPending
        AND NOT xWaitForExitClear;
END_IF

// A fault removes every externally advertised transaction signal.
IF xFaulted THEN
    xBusy := FALSE;
    xPairReq := FALSE;
    xReady := FALSE;
END_IF

END_FUNCTION_BLOCK

// Device/Application/POUs/FB_MachiningCell
FUNCTION_BLOCK FB_MachiningCell
VAR_INPUT
    tEmitterPulse   : TIME := T#500MS;
    tFeedTimeout    : TIME := T#20S;
    tPickupTimeout  : TIME := T#20S;
    tProcessTimeout : TIME := T#60S;
    xAtEntry        : BOOL;
    xAtExit         : BOOL;
    xCenterBusy     : BOOL;
    xCenterHasError : BOOL;
    xCenterOpened   : BOOL;
    xEnable         : BOOL;
    xProduceLids    : BOOL;
    xRequest        : BOOL;
    xReset          : BOOL;
    xRun            : BOOL;
END_VAR

VAR_OUTPUT
    diCount                : DINT;
    eState                 : E_MachiningCellState :=
                                 E_MachiningCellState.Stopped;
    uiFaultCode            : UINT;
	xBusy 				   : BOOL;
    xCenterProduceCmd      : BOOL;
    xCenterResetCmd        : BOOL;
    xCenterStartCmd        : BOOL;
    xCenterStopCmd         : BOOL;
    xDone                  : BOOL;
    xEmitterCmd            : BOOL;
    xExitConveyor1Cmd      : BOOL;
    xExitConveyor2Cmd      : BOOL;
    xFaulted               : BOOL;
    xRawConveyorCmd        : BOOL;
    xReady                 : BOOL;
END_VAR

VAR
    fbEmitterPulse  : TP;
    fbFeedTimeout   : TON;
    fbPickupTimeout : TON;
    fbProcessTimeout : TON;
    xEmitterIssued  : BOOL;
END_VAR

// =============================================================
// TIMERS
// Controlled Stops pause every timeout.
// =============================================================

fbEmitterPulse(
    IN :=
        xEnable
        AND xRun
        AND NOT xEmitterIssued
        AND
        (eState = E_MachiningCellState.FeedingRaw)
        AND NOT xAtEntry,
    PT := tEmitterPulse
);

fbFeedTimeout(
    IN :=
        xEnable
        AND xRun
        AND
        (eState = E_MachiningCellState.FeedingRaw)
        AND NOT xAtEntry,
    PT := tFeedTimeout
);

fbPickupTimeout(
    IN :=
        xEnable
        AND xRun
        AND
        (eState = E_MachiningCellState.WaitingForPickup)
        AND NOT xCenterBusy,
    PT := tPickupTimeout
);

fbProcessTimeout(
    IN :=
        xEnable
        AND xRun
        AND
        (eState = E_MachiningCellState.Processing)
        AND NOT xAtExit,
    PT := tProcessTimeout
);


// =============================================================
// SAFE OUTPUT DEFAULTS
// =============================================================

xCenterProduceCmd := xEnable AND xProduceLids;
xCenterResetCmd := xReset;
xCenterStartCmd := FALSE;
xCenterStopCmd :=
    (NOT xEnable OR NOT xRun OR xFaulted)
    AND NOT xReset;

xDone := FALSE;
xEmitterCmd := FALSE;
xExitConveyor1Cmd := FALSE;
xExitConveyor2Cmd := FALSE;
xRawConveyorCmd := FALSE;
xReady := FALSE;


// =============================================================
// ONE-PART EMITTER MEMORY
// =============================================================

IF fbEmitterPulse.Q THEN
    xEmitterIssued := TRUE;
END_IF

// Entry detection proves that the emitted blank arrived.
IF xAtEntry THEN
    xEmitterIssued := FALSE;
END_IF


// =============================================================
// RESET, FAULT AND RUN PRIORITIES
// =============================================================

IF xReset THEN
    diCount := 0;
    eState := E_MachiningCellState.Stopped;
    uiFaultCode := 0;
    xEmitterIssued := FALSE;
    xFaulted := FALSE;

ELSIF xCenterHasError THEN
    uiFaultCode := 100;
    xFaulted := TRUE;
    eState := E_MachiningCellState.Faulted;

ELSIF xFaulted THEN
    eState := E_MachiningCellState.Faulted;

// A controlled Stop preserves eState and xEmitterIssued.
ELSIF xEnable AND xRun THEN

    // Carry the finished item towards its exit staging sensor.
	// Stop there so the pair diverter owns the downstream release.
	xExitConveyor1Cmd :=
		(eState = E_MachiningCellState.Processing)
		AND NOT xAtExit;
	
	xExitConveyor2Cmd :=
		(eState = E_MachiningCellState.Processing)
		AND NOT xAtExit;

    CASE eState OF

        E_MachiningCellState.Stopped:
            eState := E_MachiningCellState.Ready;


        E_MachiningCellState.Ready:
            xReady :=
                xCenterOpened
                AND NOT xAtExit
                AND NOT xCenterBusy;

            IF xRequest AND xReady THEN
                eState := E_MachiningCellState.FeedingRaw;
            END_IF


        E_MachiningCellState.FeedingRaw:
            xEmitterCmd := fbEmitterPulse.Q;
            xRawConveyorCmd := TRUE;

            IF xAtEntry THEN
                eState :=
                    E_MachiningCellState.WaitingForPickup;

            ELSIF fbFeedTimeout.Q THEN
                uiFaultCode := 101;
                xFaulted := TRUE;
                eState := E_MachiningCellState.Faulted;
            END_IF


        E_MachiningCellState.WaitingForPickup:
            xCenterStartCmd := TRUE;
            xRawConveyorCmd := TRUE;

            IF xCenterBusy THEN
                eState := E_MachiningCellState.Processing;

            ELSIF fbPickupTimeout.Q THEN
                uiFaultCode := 102;
                xFaulted := TRUE;
                eState := E_MachiningCellState.Faulted;
            END_IF


        E_MachiningCellState.Processing:
            IF xAtExit THEN
                diCount := diCount + 1;
                eState := E_MachiningCellState.Complete;

            ELSIF fbProcessTimeout.Q THEN
                uiFaultCode := 103;
                xFaulted := TRUE;
                eState := E_MachiningCellState.Faulted;
            END_IF


        E_MachiningCellState.Complete:
            // Hold completion until the unit removes its request
            // and the finished product physically leaves staging.
            xDone := TRUE;

            IF NOT xRequest AND NOT xAtExit THEN
                eState := E_MachiningCellState.Ready;
            END_IF


        E_MachiningCellState.Faulted:
            xFaulted := TRUE;


    ELSE
        uiFaultCode := 199;
        xFaulted := TRUE;
        eState := E_MachiningCellState.Faulted;

    END_CASE
END_IF


// =============================================================
// FINAL COMMAND INTERLOCKS
// =============================================================

IF xFaulted THEN
    xCenterStartCmd := FALSE;
    xCenterStopCmd := NOT xReset;
    xEmitterCmd := FALSE;
    xExitConveyor1Cmd := FALSE;
    xExitConveyor2Cmd := FALSE;
    xRawConveyorCmd := FALSE;
END_IF

// Reset must never compete with Start or Stop.
IF xReset THEN
    xCenterResetCmd := TRUE;
    xCenterStartCmd := FALSE;
    xCenterStopCmd := FALSE;
END_IF

// State-derived status remains valid during a controlled Stop.
xBusy :=
    (eState = E_MachiningCellState.FeedingRaw)
    OR
    (eState = E_MachiningCellState.WaitingForPickup)
    OR
    (eState = E_MachiningCellState.Processing)
    OR
    (eState = E_MachiningCellState.Complete);

END_FUNCTION_BLOCK
